FUNCTION_BLOCK Cylinder IMPLEMENTS ICylinder
VAR_INPUT
END_VAR
VAR_OUTPUT
END_VAR
VAR
END_VAR

{warning 'add method implementation '}
METHOD bwd
END_METHOD

{warning 'add method implementation '}
METHOD fwd
END_METHOD

END_FUNCTION_BLOCK

(* stored: Version 1.1.0.1, ProductVersion 3.1.4024.12
   POU Cylinder: Id {bc59d3bc-be40-4414-9339-2d408c7d5472}, SpecialFunc None
   Method bwd: Id {7c9260b8-a926-4a28-81bb-fc0c897f9b1e}
   Method fwd: Id {5c39f43c-1f26-482b-8b91-af06775dee77} *)
